FUNCTION FuzzyNOT : REAL
VAR_INPUT
	MD:REAL;//MEMBERSHIP DEGREE
END_VAR
VAR
END_VAR

FuzzyNOT:=1-MD;

END_FUNCTION

(* stored: Version 1.1.0.1, ProductVersion 3.1.4024.6
   POU FuzzyNOT: Id {17055457-a70b-4efc-a9d6-8d2632a83c74}, SpecialFunc None *)
